{attribute 'GeneratedUsingTerminal: EL6001-0000-0020'}
{attribute addProperty BoxType "EL6001-0000-0020"}
{attribute addProperty Id "EtcSlaveTerminalBaseInputsAT %I*Inputs_37C8E74C6OutputsAT %Q*Outputs_2CF06B6A6WcStateAT %I*WcState_9091E0EB2InfoDataAT %I*InfoData_32EB74EA10"}
{attribute addProperty CRC "2312832851"}
{attribute addProperty Size "24"}
TYPE EL6001_89DB0753 EXTENDS EtcSlaveTerminalBase :
STRUCT
	{attribute addProperty Name "Inputs"}
	Inputs : Inputs_37C8E74C;
	{attribute addProperty Name "Outputs"}
	Outputs : Outputs_2CF06B6A;
	{attribute addProperty Name "WcState"}
	WcState : WcState_9091E0EB;
	{attribute addProperty Name "InfoData"}
	InfoData : InfoData_32EB74EA;
END_STRUCT
END_TYPE

(* stored: Version 1.2.0.0, ProductVersion 3.1.4024.9
   DUT EL6001_89DB0753: Id {cc4cbcdd-57e2-4817-b809-5185449c678a} *)
